// TIA Portal V17 export
// export: Created 2025-06-26T06:49:09.3089636Z, ExportSetting WithDefaults, DisplayName Totally Integrated Automation Portal, DisplayVersion V17 Update 8, DisplayName TIA Portal Openness, DisplayVersion V17 Update 8, DisplayName TIA Portal Version Control Interface, DisplayVersion V17, DisplayName STEP 7 Professional, DisplayVersion V17 Update 8, DisplayName STEP 7 Safety, DisplayVersion V17 Update 6, DisplayName WinCC Advanced, DisplayVersion V17 Update 8
FUNCTION_BLOCK "Cloud"   // FB4, FBD
TITLE = Cloud tasks
{ S7_Optimized_Access := 'TRUE' }
VERSION : 0.1
// stored: AutoNumber true, IsIECCheckEnabled false, IsRetainMemResEnabled false, MemoryReserve 0, SetENOAutomatically false, UDAEnableTagReadback false
   VAR
      CurrentTime { ExternalWritable := 'False'} : DTL;
      SetTime : DTL;
      Update : Bool;
   END_VAR
   VAR_TEMP
      ReadStatus : Int;
      WriteStatus : Int;
   END_VAR
   VAR_TEMP   // added for the SCL form of the ladder/FBD networks
      _w1 : Bool;
   END_VAR
BEGIN

REGION Network 1: Read PLC clock
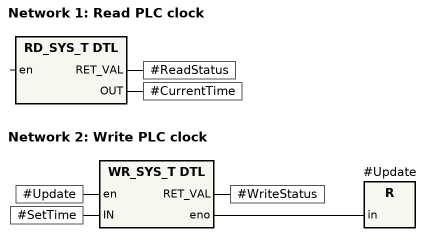
   #ReadStatus := RD_SYS_T(OUT => #CurrentTime);
END_REGION

REGION Network 2: Write PLC clock
   #WriteStatus := WR_SYS_T(EN := #Update, IN := #SetTime, ENO => #_w1);
   IF #_w1 THEN #Update := FALSE; END_IF;
END_REGION

REGION Network 3 (SCL): Manually copy interesting values to its own DB
   // This prevents messing up OPC UA URIs every time something unrelated in the program changes
   // AI
   "DB_Cloud".HBL_TT_502 := "DB_Heatbooster".AI.HBL_TT_502.fValue;
   "DB_Cloud".HBL_PT_503 := "DB_Heatbooster".AI.HBL_PT_503.fValue;
   "DB_Cloud".HBL_TT_504 := "DB_Heatbooster".AI.HBL_TT_504.fValue;
   "DB_Cloud".HBL_LT_510 := "DB_Heatbooster".AI.HBL_LT_510.fValue;
   "DB_Cloud".HBL_PT_511 := "DB_Heatbooster".AI.HBL_PT_511.fValue;
   "DB_Cloud".HBL_TT_512 := "DB_Heatbooster".AI.HBL_TT_512.fValue;
   "DB_Cloud".HBL_TT_516 := "DB_Heatbooster".AI.HBL_TT_516.fValue;
   "DB_Cloud".HBL_PT_517 := "DB_Heatbooster".AI.HBL_PT_517.fValue;
   "DB_Cloud".HBL_TT_518 := "DB_Heatbooster".AI.HBL_TT_518.fValue;
   "DB_Cloud".HBL_PT_519 := "DB_Heatbooster".AI.HBL_PT_519.fValue;
   "DB_Cloud".HBL_FT_520 := "DB_Heatbooster".AI.HBL_FT_520.fValue;
   "DB_Cloud".HBL_TT_530 := "DB_Heatbooster".AI.HBL_TT_530.fValue;
   "DB_Cloud".HBL_PT_531 := "DB_Heatbooster".AI.HBL_PT_531.fValue;
   "DB_Cloud".HBL_TT_532 := "DB_Heatbooster".AI.HBL_TT_532.fValue;
   "DB_Cloud".HBL_TT_533 := "DB_Heatbooster".AI.HBL_TT_533.fValue;
   "DB_Cloud".HBL_PT_534 := "DB_Heatbooster".AI.HBL_PT_534.fValue;
   "DB_Cloud".HBL_AT_535 := "DB_Heatbooster".AI.HBL_AT_535.fValue;
   "DB_Cloud".HBL_TT_540 := "DB_Heatbooster".AI.HBL_TT_540.fValue;
   "DB_Cloud".HBL_PT_541 := "DB_Heatbooster".AI.HBL_PT_541.fValue;
   "DB_Cloud".HBL_TT_542 := "DB_Heatbooster".AI.HBL_TT_542.fValue;
   "DB_Cloud".HBL_TT_543 := "DB_Heatbooster".AI.HBL_TT_543.fValue;
   "DB_Cloud".HBL_PT_544 := "DB_Heatbooster".AI.HBL_PT_544.fValue;
   "DB_Cloud".HBL_AT_545 := "DB_Heatbooster".AI.HBL_AT_545.fValue;
   "DB_Cloud".HBL_TT_546 := "DB_Heatbooster".AI.HBL_TT_546.fValue;
   "DB_Cloud".HBL_PT_547 := "DB_Heatbooster".AI.HBL_PT_547.fValue;
   "DB_Cloud".HBL_TT_571 := "DB_Heatbooster".AI.HBL_TT_571.fValue;
   "DB_Cloud".HBL_PT_572 := "DB_Heatbooster".AI.HBL_PT_572.fValue;
   "DB_Cloud".HBL_TT_573 := "DB_Heatbooster".AI.HBL_TT_573.fValue;
   "DB_Cloud".HBL_LT_610 := "DB_Heatbooster".AI.HBL_LT_610.fValue;
   "DB_Cloud".HBL_TT_611 := "DB_Heatbooster".AI.HBL_TT_611.fValue;
   "DB_Cloud".HBL_PT_612 := "DB_Heatbooster".AI.HBL_PT_612.fValue;
   "DB_Cloud".HBL_CT_615 := "DB_Heatbooster".AI.HBL_CT_615.fValue;
   "DB_Cloud".HBL_PT_618 := "DB_Heatbooster".AI.HBL_PT_618.fValue;
   "DB_Cloud".HBL_PT_635 := "DB_Heatbooster".AI.HBL_PT_635.fValue;
   "DB_Cloud".HBL_PT_636 := "DB_Heatbooster".AI.HBL_PT_636.fValue;
   "DB_Cloud".HBL_LT_650 := "DB_Heatbooster".AI.HBL_LT_650.fValue;
   "DB_Cloud".HBL_PT_651 := "DB_Heatbooster".AI.HBL_PT_651.fValue;
   "DB_Cloud".HBL_PT_701 := "DB_Heatbooster".AI.HBL_PT_701.fValue;
   "DB_Cloud".HBL_PT_702 := "DB_Heatbooster".AI.HBL_PT_702.fValue;
   "DB_Cloud".HBL_PT_703 := "DB_Heatbooster".AI.HBL_PT_703.fValue;
   "DB_Cloud".CPC_LT_870 := "DB_Heatbooster".AI.CPC_LT_870.fValue;
   "DB_Cloud".CPC_TT_871 := "DB_Heatbooster".AI.CPC_TT_871.fValue;
   "DB_Cloud".CPC_PT_872 := "DB_Heatbooster".AI.CPC_PT_872.fValue;
   "DB_Cloud".CPC_PT_862 := "DB_Heatbooster".AI.CPC_PT_862.fValue;
   "DB_Cloud".HBL_TT_901 := "DB_Heatbooster".AI.HBL_TT_901.fValue;
   "DB_Cloud".HBL_PT_902 := "DB_Heatbooster".AI.HBL_PT_902.fValue;
   "DB_Cloud".HBL_TT_03  := "DB_Heatbooster".AI.HBL_TT_03.fValue;
   "DB_Cloud".HBL_TT_16  := "DB_Heatbooster".AI.HBL_TT_16.fValue;
   "DB_Cloud".HBL_TT_17  := "DB_Heatbooster".AI.HBL_TT_17.fValue;
   "DB_Cloud".HBL_TT_18  := "DB_Heatbooster".AI.HBL_TT_18.fValue;
   "DB_Cloud".HBL_TT_20  := "DB_Heatbooster".AI.HBL_TT_20.fValue;
   "DB_Cloud".HBL_TT_21  := "DB_Heatbooster".AI.HBL_TT_21.fValue;
   "DB_Cloud".HBL_TT_22  := "DB_Heatbooster".AI.HBL_TT_22.fValue;
   "DB_Cloud".HBL_TT_23  := "DB_Heatbooster".AI.HBL_TT_23.fValue;
   "DB_Cloud".HBL_TT_24  := "DB_Heatbooster".AI.HBL_TT_24.fValue;
   "DB_Cloud".HBL_TT_25  := "DB_Heatbooster".AI.HBL_TT_25.fValue;
   "DB_Cloud".HBL_TT_26  := "DB_Heatbooster".AI.HBL_TT_26.fValue;
   "DB_Cloud".HBL_TT_27  := "DB_Heatbooster".AI.HBL_TT_27.fValue;
   "DB_Cloud".HBL_PT_05  := "DB_Heatbooster".AI.HBL_PT_05.fValue;
   "DB_Cloud".HBL_PT_06  := "DB_Heatbooster".AI.HBL_PT_06.fValue;
   "DB_Cloud".HBL_PT_17  := "DB_Heatbooster".AI.HBL_PT_17.fValue;
   "DB_Cloud".HBL_CT_01  := "DB_Heatbooster".AI.HBL_CT_01.fValue;
   "DB_Cloud".HBL_CT_03  := "DB_Heatbooster".AI.HBL_CT_03.fValue;
   "DB_Cloud".SSC_TT_01  := "DB_Heatbooster".AI.SSC_TT_01.fValue;
   "DB_Cloud".SSC_TT_02  := "DB_Heatbooster".AI.SSC_TT_02.fValue;
   "DB_Cloud".SSC_TT_03  := "DB_Heatbooster".AI.SSC_TT_03.fValue;
   "DB_Cloud".SSC_TT_04  := "DB_Heatbooster".AI.SSC_TT_04.fValue;
   "DB_Cloud".SSC_PIT_01 := "DB_Heatbooster".AI.SSC_PIT_01.fValue;
   "DB_Cloud".SSC_PDT_01 := "DB_Heatbooster".AI.SSC_PDT_01.fValue;
   "DB_Cloud".SSC_LT_01  := "DB_Heatbooster".AI.SSC_LT_01.fValue;
   "DB_Cloud".HBL_VT_01 := "DB_Heatbooster".AI.HBL_VT_01.fValue;
   "DB_Cloud".HBL_TT_36 := "DB_Heatbooster".AI.HBL_TT_36.fValue;

   // Calc
   "DB_Cloud".Compressor_CrankcaseSaturationTemperature := "DB_Heatbooster".Calc.Compressor.CrankcaseSaturationTemperature.fValue;
   "DB_Cloud".Compressor_CrankcaseSuperheat := "DB_Heatbooster".Calc.Compressor.CrankcaseSuperheat.fValue;
   "DB_Cloud".Compressor_VolumetricEfficiency := "DB_Heatbooster".Calc.Compressor.VolumetricEfficiency.fValue;
   "DB_Cloud".Compressor_IsentropicEfficiency := "DB_Heatbooster".Calc.Compressor.IsentropicEfficiency.fValue;
   "DB_Cloud".Compressor_Massflow := "DB_Heatbooster".Calc.Compressor.Massflow.fValue;
   "DB_Cloud".HeatSink_DeltaT := "DB_Heatbooster".Calc.HeatSink.DeltaT.fValue;
   "DB_Cloud".HeatSink_Pinch := "DB_Heatbooster".Calc.HeatSink.Pinch.fValue;
   "DB_Cloud".HeatSink_HeatRate := "DB_Heatbooster".Calc.HeatSink.HeatRate.fValue;
   "DB_Cloud".HeatSink_DeltaP := "DB_Heatbooster".Calc.HeatSink.DeltaP.fValue;
   "DB_Cloud".HeatSink_Massflow := "DB_Heatbooster".Calc.HeatSink.Massflow.fValue;
   "DB_Cloud".HeatSource_DeltaT := "DB_Heatbooster".Calc.HeatSource.DeltaT.fValue;
   "DB_Cloud".HeatSource_Pinch := "DB_Heatbooster".Calc.HeatSource.Pinch.fValue;
   "DB_Cloud".HeatSource_HeatRate := "DB_Heatbooster".Calc.HeatSource.HeatRate.fValue;
   "DB_Cloud".HeatSource_DeltaP := "DB_Heatbooster".Calc.HeatSource.DeltaP.fValue;
   "DB_Cloud".HeatSource_TemperatureRateOfChange := "DB_Heatbooster".Calc.HeatSource.TemperatureRateOfChange.fValue;
   "DB_Cloud".HeatSource_Massflow := "DB_Heatbooster".Calc.HeatSource.Massflow.fValue;
   "DB_Cloud".HighPressPart_CompressorSaturationTemperature := "DB_Heatbooster".Calc.HighPressPart.CompressorSaturationTemperature.fValue;
   "DB_Cloud".HighPressPart_CompressorSuperheat := "DB_Heatbooster".Calc.HighPressPart.CompressorSuperheat.fValue;
   "DB_Cloud".HighPressPart_CondenserSaturationTemperature := "DB_Heatbooster".Calc.HighPressPart.CondenserSaturationTemperature.fValue;
   "DB_Cloud".HighPressPart_CondenserSubcooling := "DB_Heatbooster".Calc.HighPressPart.CondenserSubcooling.fValue;
   "DB_Cloud".HighPressPart_ExpansionValveSubcooling := "DB_Heatbooster".Calc.HighPressPart.ExpansionValveSubcooling.fValue;
   "DB_Cloud".HighPressPart_CondenserDeltaP := "DB_Heatbooster".Calc.HighPressPart.CondenserDeltaP.fValue;
   "DB_Cloud".LowPressPart_EvaporatorSuperheat := "DB_Heatbooster".Calc.LowPressPart.EvaporatorSuperheat.fValue;
   "DB_Cloud".LowPressPart_CompressorSuperheat := "DB_Heatbooster".Calc.LowPressPart.CompressorSuperheat.fValue;
   "DB_Cloud".LowPressPart_EvaporatorSaturationTemperature := "DB_Heatbooster".Calc.LowPressPart.EvaporatorSaturationTemperature.fValue;
   "DB_Cloud".LowPressPart_CompressorSaturationTemperature := "DB_Heatbooster".Calc.LowPressPart.CompressorSaturationTemperature.fValue;
   "DB_Cloud".System_Quality := "DB_Heatbooster".Calc.System.Quality.fValue;
   "DB_Cloud".System_COP := "DB_Heatbooster".Calc.System.COP.fValue;
   "DB_Cloud".System_ElectricalPower := "DB_Heatbooster".Calc.System.ElectricalPower.fValue;
   "DB_Cloud".System_TemperatureLift := "DB_Heatbooster".Calc.System.TemperatureLift.fValue;
   "DB_Cloud".System_MotorEfficiency := "DB_Heatbooster".Calc.System.MotorEfficiency.fValue;
   "DB_Cloud".System_FMEP := "DB_Heatbooster".Calc.System.FMEP.fValue;
   "DB_Cloud".Auxiliary_ShaftSealDeltaT := "DB_Heatbooster".Calc.Auxiliary.ShaftSealDeltaT.fValue;
   "DB_Cloud".Auxiliary_CPCPumpDeltaP := "DB_Heatbooster".Calc.Auxiliary.CPCPumpDeltaP.fValue;
   "DB_Cloud".Misc_OilFilterDeltaP := "DB_Heatbooster".Calc.Misc.OilFilterDeltaP.fValue;

   // DI
   "DB_Cloud".HBL_FS_01 := "DB_Heatbooster".DI.HBL_FS_01;
   "DB_Cloud".HBL_FS_02 := "DB_Heatbooster".DI.HBL_FS_02;
   "DB_Cloud".HBL_LS_632 := "DB_Heatbooster".DI.HBL_LS_632;
   "DB_Cloud".HBL_LS_633 := "DB_Heatbooster".DI.HBL_LS_633;
   "DB_Cloud".CPC_LS_864 := "DB_Heatbooster".DI.CPC_LS_864;
   "DB_Cloud".VPNUserConnected := "DB_Heatbooster".DI.VPNUserConnected;

   // DO
   "DB_Cloud".HBL_EC_01 := "DB_Heatbooster".DO.HBL_EC_01;
   "DB_Cloud".HBL_EC_02 := "DB_Heatbooster".DO.HBL_EC_02;
   "DB_Cloud".HBL_HV_630 := "DB_Heatbooster".DO.HBL_HV_630;
   "DB_Cloud".HBL_HV_631 := "DB_Heatbooster".DO.HBL_HV_631;
   "DB_Cloud".HBL_HV_860 := "DB_Heatbooster".DO.HBL_HV_860;
   "DB_Cloud".HBL_HV_861 := "DB_Heatbooster".DO.HBL_HV_861;
   "DB_Cloud".SSC_P_01 := "DB_Heatbooster".DO.SSC_P_01;
   "DB_Cloud".SSC_F_01 := "DB_Heatbooster".DO.SSC_F_01;
   "DB_Cloud".SSC_P_02 := "DB_Heatbooster".DO.SSC_P_02;
   "DB_Cloud".CPC_P_01 := "DB_Heatbooster".DO.CPC_P_01;

   // Inverter
   "DB_Cloud".HBL_SC_01_A1 := "DB_Heatbooster".Inverter.HBL_SC_01_A1.fValue;
   "DB_Cloud".HBL_SC_01_A2 := "DB_Heatbooster".Inverter.HBL_SC_01_A2.fValue;
   "DB_Cloud".HBL_SC_01_A3 := "DB_Heatbooster".Inverter.HBL_SC_01_A3.fValue;
   "DB_Cloud".HBL_SC_02_A1 := "DB_Heatbooster".Inverter.HBL_SC_02_A1.fValue;
   "DB_Cloud".HBL_SC_02_A2 := "DB_Heatbooster".Inverter.HBL_SC_02_A2.fValue;
   "DB_Cloud".HBL_SC_02_A3 := "DB_Heatbooster".Inverter.HBL_SC_02_A3.fValue;
   "DB_Cloud".HBL_SC_03_A1 := "DB_Heatbooster".Inverter.HBL_SC_03_A1.fValue;
   "DB_Cloud".HBL_SC_03_A2 := "DB_Heatbooster".Inverter.HBL_SC_03_A2.fValue;
   "DB_Cloud".HBL_SC_03_A3 := "DB_Heatbooster".Inverter.HBL_SC_03_A3.fValue;
   "DB_Cloud".HBL_SC_10_A1 := "DB_Heatbooster".Inverter.HBL_SC_10_A1.fValue;
   "DB_Cloud".HBL_SC_10_A2 := "DB_Heatbooster".Inverter.HBL_SC_10_A2.fValue;
   "DB_Cloud".HBL_SC_10_A3 := "DB_Heatbooster".Inverter.HBL_SC_10_A3.fValue;

   // Valves
   "DB_Cloud".HBL_HCV_576_A1 := "DB_Heatbooster".Valve.HBL_HCV_576_A1.fValue;
   "DB_Cloud".HBL_HCV_578_A1 := "DB_Heatbooster".Valve.HBL_HCV_578_A1.fValue;
   "DB_Cloud".HBL_HCV_577_A1 := "DB_Heatbooster".Valve.HBL_HCV_577_A1.fValue;
   "DB_Cloud".HBL_HCV_579_A1 := "DB_Heatbooster".Valve.HBL_HCV_579_A1.fValue;
   "DB_Cloud".HBL_HCV_515_A1 := "DB_Heatbooster".Valve.HBL_HCV_515_A1.fValue;
   "DB_Cloud".HBL_HCV_575_A1 := "DB_Heatbooster".Valve.HBL_HCV_575_A1.fValue;
   "DB_Cloud".HBL_HCV_616_A1 := "DB_Heatbooster".Valve.HBL_HCV_616_A1.fValue;
   "DB_Cloud".HBL_HCV_700_A1 := "DB_Heatbooster".Valve.HBL_HCV_700_A1.fValue;
   "DB_Cloud".HBL_HCV_514_A1 := "DB_Heatbooster".Valve.HBL_HCV_514_A1.fValue;
   "DB_Cloud".HBL_HCV_548_A1 := "DB_Heatbooster".Valve.HBL_HCV_548_A1.fValue;

   // Other
   "DB_Cloud".ClientID := "DB_System".ClientID;
   "DB_Cloud".RunningTimeHours := "DB_Application".FromHB.RunningTimeHours;
   "DB_Cloud".RunningTimeMinutes := "DB_Application".FromHB.RunningTimeMinutes;
   "DB_Cloud".RunningTimeSeconds := "DB_Application".FromHB.RunningTimeSeconds;
   "DB_Cloud".MachineState := "DB_Application".FromHB.MachineState;
END_REGION
END_FUNCTION_BLOCK
